Staubli VAL3: motionBuffer.pgx

public program motionBuffer(num x_nMovePts, num x_nElems)
begin

  // update motion buffer size

  gotoxy(scMonitor, 0,4)
  put(scMonitor, "Motion buffer:")
  gotoxy(scMonitor, 19,4)
  put(scMonitor, x_nElems)
  gotoxy(scMonitor, 24,4)
  put(scMonitor, x_nMovePts)

end
